// TwinCAT 3 PLC project Untitled1
// ProgramVersion: 3.1.4024.0
// libraries:
//   Tc2_Standard, * (Beckhoff Automation GmbH)
//   Tc2_System, * (Beckhoff Automation GmbH)
//   Tc3_Module, * (Beckhoff Automation GmbH)
//   Tc3_Vision, * (Beckhoff Automation GmbH)
// project tree:
//   / PlcTask.TcTTO
//   POUs/ FindContoursByColour.TcPOU, Hough_1.TcPOU, MAIN.TcPOU
// real-time tasks:
//   TASK PlcTask: cycle T#150ms, priority 20, ADS port 350
//   TASK VnTask ImgAcq (FileSource1): cycle T#10ms, priority 5, ADS port 351
//   TASK JobTask1: cycle default, priority 1
//   TASK JobTask2: cycle default, priority 2
//   TASK JobTask3: cycle default, priority 3
//   TASK JobTask4: cycle default, priority 4

CONFIGURATION Untitled1
    RESOURCE PLC ON TwinCAT3
        TASK PlcTask(INTERVAL := T#150ms, PRIORITY := 20);
        PROGRAM MAIN WITH PlcTask : MAIN;
    END_RESOURCE
END_CONFIGURATION

// ---- POUs/MAIN.TcPOU
PROGRAM MAIN
VAR
	//Camera or file source
	hr: HRESULT;
	fbCamera: FB_VN_SimpleCameraControl;
	eState: ETcVnCameraState;	

	Hough: Hough_1();
	FindContoursByColour: FindContoursByColour();
END_VAR

//Hough(hr:=hr, fbCamera:=fbCamera, eState:=eState);
FindContoursByColour(hr:=hr, fbCamera:=fbCamera, eState:=eState);

END_PROGRAM

// ---- POUs/Hough_1.TcPOU
FUNCTION_BLOCK Hough_1
VAR_INPUT
		//Camera or file source
	hr: REFERENCE TO HRESULT;
	fbCamera: REFERENCE TO FB_VN_SimpleCameraControl;
	eState: REFERENCE TO ETcVnCameraState;
END_VAR
VAR_OUTPUT
END_VAR
VAR


//Images for realtime work
	ipImageIn: ITcVnImage;
	ipImageGrey: ITcVnImage;
	ipCanny:ITcVnImage;
	
// Watchdog
	hrWD 					:	HRESULT;
	tWDStop					:	DINT := 100000;	(* Stop time in us *)
	tRest 					:	DINT;
	nFunctionsMonitored		:	ULINT;
	nFractionProcessed 		:	UDINT;	
	tDuration 				:	DINT;
	
// Gaussian Filter	//iipImageSmoothed	:	ITcVnImage;
	ipImageSmoothedDisp	:	ITcVnDisplayableImage;
	ipImageSmoothed		:	ITcVnImage;
	nFilterWidth	:	UDINT	:=	7;
	nFilterHeight	:	UDINT	:=	7;

//Displayable images (for ADS Image watch and TwinCAT HMI
	ipImageInDisp: ITcVnDisplayableImage;
	ipImageGreyDisp:	ITcVnDisplayableImage;
	ipCannyDisp:	ITcVnDisplayableImage;

//Hough Circles algorithm
	ipCircles: ITcVnContainer;
	fInvAccuRatio: LREAL:= 2;
	fMinDist: LREAL:= 1000;
	eHoughMethod  : ETcVnHoughMethod:=TCVN_HM_GRADIENT ;
    fParam1       : LREAL:=  200;
    fParam2 : LREAL:=100;
    nMinRadius    : UDINT:=300;
    nMaxRadius    : UDINT:=400;
	
//Loop to interate through found circles
	ipIteratorCircles: 	ITcVnForwardIterator;	
	nCircles: ULINT;
	iCircle: ULINT;
	currentCircle: TcVnVector3_REAL;

//Draw
	aColorRed	: TcVnVector4_LREAL:= [255,0,0,0];
	aColorBlue	: TcVnVector4_LREAL:= [0,0,255,0];	

END_VAR

eState:= fbCamera.GetState();

IF eState = TCVN_CS_ERROR THEN
	hr:= fbCamera.Reset();
	
ELSIF eState<TCVN_CS_ACQUIRING THEN
	hr:= fbCamera.StartAcquisition();
	
ELSIF eState= TCVN_CS_ACQUIRING THEN
	
	//Get the image from camera. Or in this case a file source
	// Step 1 - Import image
	hr:= fbCamera.GetCurrentImage(ipImageIn);
	
	IF SUCCEEDED(hr) AND ipImageIn <> 0 THEN
	
	//Colour to Grey image	
		hr:= F_VN_ConvertColorSpace(ipImageIn, ipImageGrey, TCVN_CST_RGB_TO_GRAY, hr);
		
		//Start watchdog to limit the time allowed for the functions below. 
		hrWD := F_VN_StartRelWatchdog(tWDStop, hr);
	
	//Filter image smooth. Otherwise there will be a lot of false circles found
	hr:= F_VN_GaussianFilter(ipImageGrey, ipImageSmoothed, nFilterWidth, nFilterHeight, hr);

	//Call the Method Canny just for demonstration purposes to see what is output from the Canny Edge detector that is otherwise built in to the HoughCirclesExp
	hr:=Canny(ipImageSmoothed,ipCanny,ipCannyDisp, hr);
	
	//Find circles in image based on Hough Transform algorithm. This algorith finds the radius(r) plus the x and y coordinates of the center point. 
	//Since all three are considered to be unknown parameters, the circle edge direction (GRADIENT) is used to make the algorithm more efficient and minimise the numbers of guesses in the accumulator matrix.  
	//F_VN_HoughCirclesExp has a built in Canny Edge detector algorithm and takes a smoothed greyscale image as input
	//fParam1,fParam2 are the upper and lower treshold for the Canny Edge detector and define what is considered to be an edge. 
	//Over the upper is and edge. Under the lower is not. In between is an edge if a neighboruing pixel is and edge.
	//For more information about how a Hough Circles or Hough Line algorithm works. Search the internet for example "Hough Circles" for a theoretical explanation or "OpenCV HoughCircles" for the code functionality. 
	//For more information on how a Canny edge detector works. Search the terms "Canny edge detector"
	hr:=F_VN_HoughCirclesExp(ipImageSmoothed,ipCircles,fInvAccuRatio, fMinDist,eHoughMethod, fParam1,fParam2, nMinRadius, nMaxRadius, hr);
	
	hr:=  hr := F_VN_GetNumberOfElements(ipCircles, nCircles, hr);
	
	//Get interator to iterate through found circles hold by the container that the pointer ipCircles point at
	hr := F_VN_GetForwardIterator(ipCircles,ipIteratorCircles,hr);

	//Get the circles radius, x and y - And draw the result in the coloured imageIn
IF SUCCEEDED(hr) AND nCircles>0 THEN
	FOR iCircle:=0 TO nCircles-1 DO
		F_VN_GetAt_TcVnVector3_REAL(ipCircles,currentCircle, iCircle,hr);  
		hr:= F_VN_DrawCircle(REAL_TO_UDINT(currentCircle[0]),REAL_TO_UDINT(currentCircle[1]), REAL_TO_UDINT(currentCircle[2]), ipImageIn,aColorRed,2, hr);
		hr:= F_VN_DrawPointExp(REAL_TO_UDINT(currentCircle[0]),REAL_TO_UDINT(currentCircle[1]), ipImageIn,1,aColorBlue,10,2,1,hr);
		hr:= F_VN_IncrementIterator(ipIteratorCircles,hr);
	END_FOR
END_IF				
		//Stop watchdog to limit the time allowed for the functions above. 
		hrWD := F_VN_StopWatchdog(hrWD, nFunctionsMonitored => nFunctionsMonitored, nFractionProcessed => nFractionProcessed, tRest => tRest);
		
		// Calculate the required time
 		tDuration := tWDStop - tRest;
	
	//Create images to display for the different processing steps
		hr:= F_VN_CopyIntoDisplayableImage(ipImageIn, ipImageInDisp, hr);   //The result is also drawn in to this image
		hr:= F_VN_CopyIntoDisplayableImage(ipImageGrey, ipImageGreyDisp, hr); 
		hr:= F_VN_CopyIntoDisplayableImage(ipImageSmoothed, ipImageSmoothedDisp, hr);  
	
	END_IF
	
END_IF

METHOD Canny : HRESULT
VAR_INPUT
	ipImageToSearchForEdges: REFERENCE TO ITcVnImage;
	ipImageResultWithEdges: REFERENCE TO ITcVnImage;
	ipImageResultWithEdgesDisp: REFERENCE TO ITcVnDisplayableImage;
	hr: REFERENCE TO HRESULT;
END_VAR
hr:= F_VN_CannyEdgeDetection(ipImageToSearchForEdges,ipImageResultWithEdges,100, 200, hr);

hr:= F_VN_CopyIntoDisplayableImage(ipImageResultWithEdges, ipImageResultWithEdgesDisp, hr);  //saädfkaöläsfaf
END_METHOD

END_FUNCTION_BLOCK

// ---- POUs/FindContoursByColour.TcPOU
FUNCTION_BLOCK FindContoursByColour
VAR_INPUT
			//Camera or file source
	hr: REFERENCE TO HRESULT;
	fbCamera: REFERENCE TO FB_VN_SimpleCameraControl;
	eState: REFERENCE TO ETcVnCameraState;
	
END_VAR
VAR_OUTPUT
END_VAR
VAR

//Images for realtime work
	ipImageIn: ITcVnImage;
	ipImageGrey: ITcVnImage;
	ipImageBinary: ITcVnImage;

	
// Watchdog
	hrWD 					:	HRESULT;
	tWDStop					:	DINT := 120000;	(* Stop time in us *)
	tRest 					:	DINT;
	nFunctionsMonitored		:	ULINT;
	nFractionProcessed 		:	UDINT;	
	tDuration 				:	DINT;
	
// Gaussian Filter	//

	ipImageSmoothed	:	ITcVnImage;
	ipImageSmoothedDisp	:	ITcVnDisplayableImage;
	nFilterWidth	:	UDINT	:=	51;
	nFilterHeight	:	UDINT	:=	51;


	
//Displayable images (for ADS Image watch and TwinCAT HMI
	ipImageInDisp: ITcVnDisplayableImage;
	ipImageGreyDisp:	ITcVnDisplayableImage;
	ipImageBinaryDisp: ITcVnDisplayableImage;
	
//Colourlimits Upper/Lower RGB-values
	aColorHi	: TcVnVector4_LREAL:= [255,200,110];
	aColorLow	: TcVnVector4_LREAL:= [200,0,0];
	
//Create Structuring element for the Closing operation
ipStructuringElement: ITcVnImage;
eShape: ETcVnStructuringElementShape :=TCVN_SES_RECTANGLE;

eOperator: ETcVnMorphologicalOperator:=TCVN_MO_CLOSING;


ipContourList: 	ITCVnContainer;
	ipIterator: 	ITcVnForwardIterator;
	ipContour:		ITcVnContainer;
	fArea:				LREAL;
	fCurrentArea: LREAL:=5000;
	antalKonturer: ULINT;	
		aCenter:		TcVnPoint2_LREAL;

//Draw
	aColorRed	: TcVnVector4_LREAL:= [255,0,0,0];
	aColorBlue	: TcVnVector4_LREAL:= [0,0,255,0];	

	nisse: INT;
	sArea: STRING;
	nArea: ULINT;
END_VAR

eState:= fbCamera.GetState();

IF eState = TCVN_CS_ERROR THEN
	hr:= fbCamera.Reset();
	
ELSIF eState<TCVN_CS_ACQUIRING THEN
	hr:= fbCamera.StartAcquisition();
	
ELSIF eState= TCVN_CS_ACQUIRING THEN
	
	//Get the image from camera. Or in this case a file source
	// Step 1 - Import image
	hr:= fbCamera.GetCurrentImage(ipImageIn);
	
	IF SUCCEEDED(hr) AND ipImageIn <> 0 THEN


	
	
	
//Start watchdog to limit the time allowed for the functions below. 
hrWD := F_VN_StartRelWatchdog(tWDStop, hr);

//Filter image smooth. Otherwise there will be a lot of false circles found
	hr:= F_VN_GaussianFilter(ipImageIn, ipImageSmoothed, nFilterWidth, nFilterHeight, hr);
	
hr:= F_VN_CopyIntoDisplayableImage(ipImageSmoothed, ipImageSmoothedDisp, hr); 

		hr:= F_VN_CheckColorRange(ipImageSmoothed, ipImageBinary, aColorLow, aColorHi, hr);
			hr:= F_VN_CreateStructuringElement(ipStructuringElement,eShape, 25, 25, hr);		
			hr:= F_VN_MorphologicalOperator(ipImageBinary, ipImageBinary, eOperator,ipStructuringElement, hr);
			//hr:= F_VN_MorphologicalOperator(ipImageBinary, ipImageBinary, TCVN_MO_EROSION,ipStructuringElement, hr);
			hr:=F_VN_FindContours(ipImageBinary, ipContourList, hr);

			hr:= F_VN_GetNumberOfElements(ipContourList,antalKonturer,hr);
		
		hr:= F_VN_GetForwardIterator(ipContourList, ipIterator, hr);  //Create iterator
		
		//Loop through every contour with the iterator
		WHILE SUCCEEDED(hr) AND_THEN ipIterator.CheckIfEnd() <> S_OK DO
			hr:= F_VN_GetContainer(ipIterator, ipContour, hr);
			hr:= F_VN_IncrementIterator(ipIterator, hr);

 			

			//Sort out only large elements
			hr:= F_VN_ContourArea(ipContour, fArea, hr);
				IF fArea > fCurrentArea THEN
					nisse:=nisse+1;
					nArea:=LREAL_TO_ULINT(fArea);
					
					sArea:=CONCAT(CONCAT('Area: ',ULINT_TO_STRING(nArea)),' pixels');
								hr:= F_VN_DrawContours(ipContour, -1, ipImageIn, aColorRed, 3, hr);
										hr:= F_VN_ContourCenterOfMass(ipContour, aCenter, hr);
										hr:= F_VN_PutTextExp(sArea,ipImageIn, LREAL_TO_UDINT(aCenter[0])-400,LREAL_TO_UDINT(aCenter[1]), ETcVnFontType.TCVN_FT_HERSHEY_PLAIN, 4, aColorRed,3,TCVN_LT_8_CONNECTED,FALSE, hr);
										//LREAL_TO_STRING(fArea)
				END_IF


				
		END_WHILE
				
//Stop watchdog to limit the time allowed for the functions above. 
hrWD := F_VN_StopWatchdog(hrWD, nFunctionsMonitored => nFunctionsMonitored, nFractionProcessed => nFractionProcessed, tRest => tRest);

hr:= F_VN_CopyIntoDisplayableImage(ipImageBinary, ipImageBinaryDisp, hr);
	hr:= F_VN_CopyIntoDisplayableImage(ipImageIn, ipImageInDisp, hr); 

END_IF
END_IF

END_FUNCTION_BLOCK
